(* IEC 61131-3 sources: windowtracking/src/Events, 3 files *)

(* ---- ITriggerEvent.st ---- *)
USING Simatic.Ax.WindowTracking.Trigger;

NAMESPACE Simatic.Ax.WindowTracking.Events
    INTERFACE ITriggerEvent
        METHOD Action : EventStatus
            VAR_INPUT
                te : IVirtualTrigger;
                tw : ITransportWindow;
            END_VAR
        END_METHOD
    END_INTERFACE

END_NAMESPACE

(* ---- ClearWindow.st ---- *)
USING Simatic.Ax.WindowTracking.Trigger;

NAMESPACE Simatic.Ax.WindowTracking.Events
    CLASS ClearWindow IMPLEMENTS ITriggerEvent
        VAR PUBLIC
            WindowList : ITransportWindowsCleanup;
        END_VAR

        METHOD PUBLIC Action : EventStatus
            VAR_INPUT
                te : IVirtualTrigger;
                tw : ITransportWindow;
            END_VAR
            // Remove oldest window from list
            WindowList.Remove();
            ;
        END_METHOD
    END_CLASS
END_NAMESPACE

(* ---- ExitPoint.st ---- *)
USING Simatic.Ax.WindowTracking.EventHandler;
USING Simatic.Ax.WindowTracking.Trigger;
USING Simatic.Ax.WindowTracking.SortDecission;

NAMESPACE Simatic.Ax.WindowTracking.Events
    CLASS ExitPoint IMPLEMENTS ITriggerEvent

        VAR PUBLIC
            SortDecission : ISortDecission;
            ExitHandler : IExitPointHandler;
        END_VAR

        METHOD PUBLIC Action : EventStatus
            VAR_INPUT
                te : IVirtualTrigger;
                tw : ITransportWindow;
            END_VAR
            VAR_TEMP
                _sortItem : BOOL;
            END_VAR
            _sortItem := SortDecission.Check(tw := tw, te := te, exitpoint := ExitHandler);

        END_METHOD

    END_CLASS
END_NAMESPACE
